FUNCTION_BLOCK FB_CameraTrigger EXTENDS FB_Commons IMPLEMENTS I_CameraTrigger, I_StartPosDetect
(*************************************************************************************************)
(*  FILENAME:    FB_CameraTrigger                                                                *)
(*  PROJECT:     CALMAR PUPLC                                                                    *)
(*  COPYRIGHT:   All rights reserved (c) Wifag//Polytype, Fribourg/Switzerland (2016)            *)
(*  ENVIRONMENT: TwinCAT PLC                                                                     *)
(*  VERSION:     <version>                                                                       *)
(*************************************************************************************************)
(*  DESCRIPTION:                                                                   <description> *)
(*    Generate timestamp trigger output based on timestamp sensor input. Two variants            *)
(*    exist, a timebased approach where the trigger time is calculated at the time the sensor    *)
(*    event occurs, and a second approach where the sensor event time is translated to a sensor  *)
(*    event position, and a trigger is generated when the calculated trigger position has almost *)
(*    been reached. The second approach has the advantage that is is less susceptible to speed   *)
(*    variations.                                                                                *)
(*                                                                                </description> *)
(*************************************************************************************************)

{library public}
VAR_INPUT
  bI_HwEnable                             : BOOL;            // relase (enable SheetDetect) from machine
  (* - (EL1252) StartPosition detect sensor*)
  bI_Sensor_State                   AT%I* : BOOL;            // Sensor signal
  tI_Sensor_TimeStampPos            AT%I* : T_DCTIME64;      // Sensor last detection timestamp
  (* - (EL1252) Camera started feedback trigger/signal*)
  bI_TriggerFeedback_State          AT%I* : BOOL;           // Sensor signal
  tI_TriggerFeedback_TimeStampPos   AT%I* : T_DCTIME64;     // Sensor last detection timestamp

  (*System signals*)
  iI_CurrentPos                   : DINT;                   // Current position in [SubPx]*)
  fI_ConveyorSpeed                : LREAL;                  // Current speed of substrate in [m/s]*)
  
  (*Exernal command*)
 // bI_ManualTeach                  : BOOL;                   // External manual teach is active

  (*Debug & Test*)
  bI_ManualTrigger                : BOOL;                   // Manual start trigger
END_VAR

VAR_OUTPUT
  (*Link to EL2252*)
  ObTrigger                 AT%Q* : BOOL;                   // EL2252 Output1 - TRUE=start camer
  OtTriggerStartTime        AT%Q* : T_DCTIME64;             // EL2252 Timestamp - where to set outputs
  OnTriggerCommand          AT%Q* : BYTE;                   // EL2252 Command - activation timestamp ouput
END_VAR

(*{library private}*)
VAR
  bInitOk                         : BOOL;           // initialized
  bSpeedValid                     : BOOL;           // speed is valid
  bTriggerArmed                   : BOOL;           // trigger is armed
  bCamValid                       : BOOL;           // camera is valid
  bTriggerOk                      : BOOL;
  rT_Sensor                       : R_TRIG;        // rising edge trigger sensor
  
  (*configuration*)
  _nResolution                    : INT := 1;       // Printhead Resolution [e.g. 600] x Subpixel Resolution [e.g. 32]*)
  _bUsePositionTrigger            : BOOL;           // FALSE: Calculate time with speed and position distance@sensor event, TRUE: Calculate sensor event position, launch trigger based on position
  _bUseCameraTrigger              : BOOL;           // (cam specific setting) Generate camera trigger output
  _bUseCameraTriggerFeedback      : BOOL;           // (cam specific setting) Evaluate camera triggered feedback
  _bCamManualTeachMode            : BOOL;           // cam in manual teach mode
  _tMemTriggerFeedback_TimeStampPos : T_DCTIME64;
  _nSubstrateLength               : DINT;           // Substrate length in pulse [SubPx]
  _fSubstrateLength               : LREAL;          // Substrate length in [m]
  _fTriggerDistance               : LREAL;          // Distance between Sensor and Trigger [m]
  _fTriggerLength                 : LREAL := 10;    // Length of trigger signal in ms, min. 3 bus cycles
  
  iActiveCam	                    : I_CameraTriggerDevice;  // active camera interface
  
  bSheetDetected                  : BOOL;
  bInhibitTrigger                 : BOOL;            (*inhibit trigger signals, TRUE=inhibit*)
  bReleaseInhibitTrigger          : BOOL;            (*condition to release inhibit trigger*)

  eState                          : BYTE;            (*State*)
  tSensor_TimeStamp               : T_DCTIME64;      (*Sensor last detection timestamp*)
  tTriggerFeedback_TimeStamp      : T_DCTIME64;      (*Trigger feedback last detection timestamp*)
  tCurrentTime                    : T_DCTIME64;      (*Current system dc time [64bit]*)
  tTrigger_EventTime              : T_DCTIME64;      (*Trigger event timestamp*)

  _bManualStart                   : BOOL;
  fDeltaDistance                  : LREAL;           (*Distance that the substrate moved between the detection and the treatment of the information [m]*)
  _nX0                            : DINT;            (*Detected X0 position of CT [SubPx] by sensor*)
  _nCamStartPos                   : DINT;            (*Camera start position*)
  _nCamStartedPos                 : DINT;            (*Camera started position [SubPx]*)
  
  tCurrentTimeStamp               : T_DCTIME64;      (* Get Current Timestamp *)
  tLastTimeStamp                  : T_DCTIME64;      (* Get Current Timestamp *)
  fCycleTime                      : LREAL;           (* Current calcualted cycle time [s]*)

  fRemDist                        : LREAL;           (*Remaining distance until trigger occurs [m]*)
  fPreTriggerPosition             : LREAL;           (*Margin between effective trigger position and generation of timestamp*)

  fb_FTrig_ManualTeach            : F_TRIG;          (*FTrig for teach to release inhibit*)
  
  (*Debug*)
  _bVerbose                       : BOOL;
END_VAR

VAR CONSTANT
  fC_MIN_CONVEYOR_SPEED           : LREAL := 0.01;
  fC_PreTrigFactor                : LREAL := 3.0;
  fC_SheetLengthMargin            : LREAL := 0.01;   (*Added 10 mm margin for substrate length in case of print quality strips at the end of sheet in case of start with edge*)
  fC_MaxCameraFeedbackTimeout     : LREAL := 28.0;   (*[ns] Max. timeout waiting for camera trigger feedback signal*)

  (*State*)
  cL_IDLE                         : BYTE := 0;       (*Idle state, no trigger active*)
  cL_SENSOREVENT                  : BYTE := 1;       (*Sensor started trigger generation*)
  cL_WAITALMOSTSTART              : BYTE := 2;       (*Wait timestamp calculation critera*)
  cL_WAITSTART                    : BYTE := 3;       (*Wait for trigger generation critera*)
  cL_WAITFEEDBACK                 : BYTE := 4;       (*Wait on feedback from trigger*)
  cL_TRIGACTIVE                   : BYTE := 5;       (*Trigger set*)
  cL_WAITSTOP                     : BYTE := 6;       (*Trigger reset*)

  (*EL2252 Command*)
  cL_INACTIVE                     : BYTE := 0;
  cL_ACTIVE                       : BYTE := 3;
END_VAR
// TODO: convert all LREAL_TO_ULINT to save functions with range overflow check (add to CalmarCommons) to prevent crashes

IF NOT bInitOk THEN RETURN; END_IF;

// General calculations
bSpeedValid   := fI_ConveyorSpeed > fC_MIN_CONVEYOR_SPEED;    // speed valid (ignore trigger if not moving)
bCamValid     := SEL(iActiveCam<>0, FALSE, TRUE);             // camera valid (ignore trigger otherwise)
tCurrentTime  := F_GetCurDcTaskTime64();                      // current dc time (most accurate time stamp we have)
fCycleTime    := (TO_LREAL(tCurrentTime) - TO_LREAL(tLastTimeStamp)) * 1E-9;  tLastTimeStamp  := tCurrentTime;  // calculate cycle time of this block
bSheetDetected:= FALSE;                                       // Set to true below just for one cycle
bTriggerArmed :=  NOT bInhibitTrigger AND bSpeedValid AND bI_HwEnable;
rT_Sensor(CLK:=bI_Sensor_State);

IF bCamValid THEN    // save dynamic changable settings
  _fTriggerDistance := iActiveCam.fTriggerDistance;
  _fTriggerLength   := iActiveCam.fTriggerPulseLength;
END_IF


(*State Machine ----------------------------------------------------------------*)
CASE eState OF
  cL_IDLE:     (*Not started, waiting for start trigger*)
  
    IF bTriggerArmed THEN (*ignore trigger else*)
 
      IF rT_Sensor.Q AND (bCamValid OR _bCamManualTeachMode) THEN      (*Start launched*)
        eState            := cL_SENSOREVENT;
        tSensor_TimeStamp := tI_Sensor_TimeStampPos;
        _bManualStart := FALSE;
        IF _bCamManualTeachMode THEN LogWarning('StartTrigger in manual teach mode'); END_IF
      ELSIF (bI_ManualTrigger AND bCamValid) THEN  (*Manual start launched*)
        eState            := cL_SENSOREVENT;
        tSensor_TimeStamp := tCurrentTime;
        _bManualStart := TRUE;
      ELSIF (rT_Sensor.Q OR bI_ManualTrigger) AND NOT bCamValid THEN   (*Trigger without active camera*)
        LogWarning('No camera or start device active, ignore trigger');
      END_IF;
      
    END_IF
    
    OnTriggerCommand := cL_INACTIVE;
    ObTrigger        := FALSE;

  cL_SENSOREVENT:     (*Not started*)
    IF NOT bSpeedValid THEN 
      eState := cL_IDLE;        // ignore trigger if not moving anymore (avoid zero division)
    ELSE
      (*Distance in [m] that the substrate has traveled between the sensor detection (time) current plc cycle*)
      fDeltaDistance     := UINT64_TO_LREAL(UInt64Sub64(ULINT_TO_ULARGE(tCurrentTime), ULINT_TO_ULARGE(tSensor_TimeStamp))) * 1E-9 * fI_ConveyorSpeed;
      (*Position where the sheet has been detected in [SubPx]*)
      _nX0               := iI_CurrentPos - F_MeterToSubPixel(fPosMeter:=fDeltaDistance, fResoSubPx:=_nResolution);
      
      IF _bUsePositionTrigger OR NOT _bUseCameraTrigger THEN
        eState             := cL_WAITALMOSTSTART;
      ELSE
        eState             := cL_WAITSTART;
        tTrigger_EventTime := (tSensor_TimeStamp + LREAL_TO_ULINT(_fTriggerDistance / fI_ConveyorSpeed * 1E9));
      END_IF;
      
      OnTriggerCommand := cL_INACTIVE;
      ObTrigger         := TRUE;
      bInhibitTrigger   := TRUE;
      bSheetDetected    := TRUE;
      
    END_IF

  cL_WAITALMOSTSTART: (*Only active when bI_UsePositionTrigger=TRUE: wait until Start position almost reached, then set timestamp*)
    (*Remaining distance in [m], converted to REAL to avoid integer wrap problems*)
    fRemDist             := _fTriggerDistance + (DINT_TO_REAL(_nX0) - DINT_TO_REAL(iI_CurrentPos))*0.0254 / INT_TO_REAL(_nResolution);
    fPreTriggerPosition  := fC_PreTrigFactor * fCycleTime * fI_ConveyorSpeed;

    IF fRemDist < fPreTriggerPosition THEN
      eState             := cL_WAITSTART;
      tTrigger_EventTime := (tSensor_TimeStamp + LREAL_TO_ULINT(fRemDist / fI_ConveyorSpeed * 1E9));    // division save because we are moving to reach this position
      IF _bUseCameraTrigger AND NOT _bManualStart THEN
        OnTriggerCommand := cL_ACTIVE;  (*Arm EL2252*)
      END_IF
      LogTsDiff(aIdent:= 'WAITALMOSTSTART: ', t1:=tTrigger_EventTime, t2:=tCurrentTime);
    ELSE
      eState           := cL_WAITALMOSTSTART;
      OnTriggerCommand := cL_INACTIVE;
    END_IF;
    ObTrigger          := TRUE;

  cL_WAITSTART:       (*Wait until start time reached*)
    bTriggerOk := TRUE;
    IF (tTrigger_EventTime < tCurrentTime) THEN (* StartTime elapsed *)
      // position reached
      IF _bUseCameraTriggerFeedback THEN
        eState         := cL_WAITFEEDBACK;
      ELSE
        eState         := cL_TRIGACTIVE;
        iActiveCam.CamTrigger(bOk:=bTriggerOk, nPos:=iI_CurrentPos, nPosDeviation:=0);
      END_IF

      OnTriggerCommand := cL_INACTIVE; (*Disarm already command to EL2252, trigger generated*)
    ELSE
      // position not yet reached
      eState           := cL_WAITSTART;
      IF _bUseCameraTrigger AND NOT _bManualStart THEN
        OnTriggerCommand := cL_ACTIVE;  (*Arm EL2252*)
      END_IF
    END_IF;

    ObTrigger      := TRUE;  
    
  cL_WAITFEEDBACK:
    IF _bManualStart THEN //Simulate feedback in case of manual start
      tTriggerFeedback_TimeStamp:= tTrigger_EventTime + LREAL_TO_ULINT(1000.0 * 1E3); //Trigger event plus 1000ns
    ELSE
      IF tI_TriggerFeedback_TimeStampPos = _tMemTriggerFeedback_TimeStampPos AND tCurrentTime > (tTrigger_EventTime + LREAL_TO_ULINT(fC_MaxCameraFeedbackTimeout * 1E3)) THEN
        // feedback was not received in next plc cycle (timeout jitter in camera max. 28us)
        LogError(F_Concat3('No Camera trigger feedback received (timeout), after ', TO_STRING(TO_LREAL(tCurrentTime-tTrigger_EventTime)/1E6), 'ms'));
        bTriggerOk := FALSE;
        tTriggerFeedback_TimeStamp:= tTrigger_EventTime + LREAL_TO_ULINT(fC_MaxCameraFeedbackTimeout * 1E3);
      ELSE
        tTriggerFeedback_TimeStamp:= tI_TriggerFeedback_TimeStampPos;
			END_IF
    END_IF
    
  (*feedback signal is a very short trigger that the PLC sometimes cannot register, therefore we use the timestamp*)
    IF (tTriggerFeedback_TimeStamp <> _tMemTriggerFeedback_TimeStampPos) AND (tTriggerFeedback_TimeStamp > 0) OR _bManualStart THEN
      eState          := cL_TRIGACTIVE;
      // start position requested
      fDeltaDistance  := UINT64_TO_LREAL(UInt64Sub64(ULINT_TO_ULARGE(tCurrentTime), ULINT_TO_ULARGE(tTrigger_EventTime))) * 1E-9 * fI_ConveyorSpeed;
      _nCamStartPos   := _nX0 +   F_MeterToSubPixel(fPosMeter:=_fTriggerDistance, fResoSubPx:=_nResolution);
      
      // effective started position
      fDeltaDistance  := UINT64_TO_LREAL(UInt64Sub64(ULINT_TO_ULARGE(tCurrentTime), ULINT_TO_ULARGE(tTriggerFeedback_TimeStamp))) * 1E-9 * fI_ConveyorSpeed;
      _nCamStartedPos := iI_CurrentPos - F_MeterToSubPixel(fPosMeter:=fDeltaDistance, fResoSubPx:=_nResolution);
      IF _bManualStart THEN iActiveCam.CamTrigger(bOk:=bTriggerOk, nPos:=_nCamStartPos, nPosDeviation:=0);
      ELSE                  iActiveCam.CamTrigger(bOk:=bTriggerOk, nPos:=_nCamStartPos, nPosDeviation:=-_nCamStartedPos+_nCamStartPos); END_IF  (*!!!!   sign inverted*)
    ELSE
     eState           := cL_WAITFEEDBACK;
    END_IF    
    
  cL_TRIGACTIVE:   (*Trigger high*)
    eState         := cL_WAITSTOP;
    
    // calculate end timestamp of trigger (end of trigger active signal)
    tTrigger_EventTime := (tTrigger_EventTime + LREAL_TO_ULINT(_fTriggerLength * 1E6));
    
    OnTriggerCommand := cL_INACTIVE;
    ObTrigger        := FALSE;
    
  cL_WAITSTOP:  (*Wait until trigger time has elapsed*)
    IF (tTrigger_EventTime < tCurrentTime) THEN (* StopTime elapsed *)
      eState           := cL_IDLE;
      OnTriggerCommand := cL_INACTIVE; (*Disarm EL2252, trigger generated*)
      iActiveCam.CamTriggerDone();
    ELSE
      eState           := cL_WAITSTOP;
      IF _bUseCameraTrigger THEN
        OnTriggerCommand := cL_ACTIVE;  (*Arm EL2252*)
      END_IF
    END_IF;

    ObTrigger        := FALSE;

  ELSE  (*Default*)
    eState           := cL_IDLE;
    ObTrigger        := FALSE;
    OnTriggerCommand := cL_INACTIVE;
END_CASE;

OtTriggerStartTime := tTrigger_EventTime;

_tMemTriggerFeedback_TimeStampPos := tI_TriggerFeedback_TimeStampPos;

(*Release inhibit trigger*)
bReleaseInhibitTrigger := (iI_CurrentPos >= (_nX0 + _nSubstrateLength));
//fb_FTrig_ManualTeach(CLK := bI_ManualTeach);

IF (bReleaseInhibitTrigger OR fb_FTrig_ManualTeach.Q) AND bInhibitTrigger THEN
	bInhibitTrigger := FALSE;
END_IF;

(********************************* END OF FB *****************************************************)

PROPERTY bManualTeach : BOOL
GET
bManualTeach := _bCamManualTeachMode;
END_GET
SET
_bCamManualTeachMode := bManualTeach;
END_SET
END_PROPERTY

(*
  A new container detected on X0.
  NOTE: a pulse only
*)
PROPERTY bStartTrig : BOOL
GET
bStartTrig := bSheetDetected;
END_GET
END_PROPERTY

(*
  A valid container detected.
*)
PROPERTY bValid : BOOL
GET
bValid := bSheetDetected AND NOT _bCamManualTeachMode AND bCamValid;  // in manual teach the ct is "present" should not be printed
END_GET
END_PROPERTY

METHOD Disable : BOOL
IF eState = cL_IDLE THEN
  iActiveCam := 0;
  Disable := TRUE;
ELSE  
  Disable := FALSE;
  LogError('disable failed: trigger busy');
END_IF
END_METHOD

METHOD Enable : BOOL
VAR_INPUT
	iCam	                    : I_CameraTriggerDevice;
  bUseCameraTrigger         : BOOL; //Generate camera trigger
  bUseCameraTriggerFeedback : BOOL; //Use feedback as trigger?
END_VAR
IF iCam = 0 THEN
  Enable := FALSE;
  LogError('setCam failed: invalid reference');
ELSIF eState <> cL_IDLE THEN
  Enable := FALSE;
  LogError('enable failed: trigger busy');
ELSE
  iActiveCam := iCam;
  Enable     := TRUE;

  // save constant settings
  _bUseCameraTrigger := bUseCameraTrigger;
  _bUseCameraTriggerFeedback := bUseCameraTriggerFeedback;
END_IF;
END_METHOD

METHOD Init
VAR_INPUT
  nResolution                   : INT := 1;        (*Printhead Resolution [e.g. 600] x Subpixel Resolution [e.g. 32]*)
  bUsePositionTrigger           : BOOL;            (*FALSE: Calculate time with speed and position distance@sensor evont*)
END_VAR
(*zero divisions*)
IF nResolution = 0 THEN 
  bInitOk :=FALSE;
  RETURN; 
END_IF;

_nResolution:=nResolution;
_bUsePositionTrigger :=bUsePositionTrigger;


bInitOk :=TRUE;
END_METHOD

(*
  Log timestamp difference (if verbose active).
  t1-t2 
*)
METHOD LogTsDiff : BOOL
VAR_INPUT
  aIdent : STRING;
  t1 : T_DCTIME64;
  t2 : T_DCTIME64;
END_VAR
IF _bVerbose THEN
  LogLvl(Lvl:=E_LogSeverity.Debug, Msg:=
       F_Concat7(aIdent, 
                 't1: ', TO_STRING(t1), 
                 ' t2: ', TO_STRING(t2), 
                 ' t1-t2 [ms]: ', TO_STRING((TO_LREAL(t1)-TO_LREAL(t2))*1E-6)
       )
  );
END_IF
END_METHOD

(*
  Detected start position X0 (absolute) in [SubPx].
*)
PROPERTY nStartPositionX0 : DINT
GET
nStartPositionX0 := _nX0;
END_GET
END_PROPERTY

METHOD Reset
VAR_INPUT
END_VAR
eState          := cL_IDLE;
bInhibitTrigger := FALSE;
END_METHOD

METHOD SetSubstrateLength
VAR_INPUT
  fSubstrateLength : LREAL;
END_VAR
IF NOT bInitOk THEN RETURN;END_IF;

(*Added 10 mm margin for substrate length in case of print quality strips at the end of sheet in case of start with edge*)
_fSubstrateLength := fSubstrateLength + fC_SheetLengthMargin;
_nSubstrateLength := F_MeterToSubPixel(fPosMeter:=_fSubstrateLength, fResoSubPx:=_nResolution);
END_METHOD

END_FUNCTION_BLOCK

(* stored: Version 1.1.0.1, ProductVersion 3.1.4024.3
   POU FB_CameraTrigger: Id {b0f3b9ca-3ef5-425e-9c4d-fa0358aa72fd}, SpecialFunc None
   Property bManualTeach: Id {58f64ca5-2fbd-4f19-9c85-e284ce94b427}
   Get Get: Id {4c3cab32-2be9-4a94-8004-e45185b9890b}
   Set Set: Id {7bf6ee58-08a2-435d-af4d-9a1743824b8f}
   Property bStartTrig: Id {744708b2-efbe-44a0-b99d-f740e061c41a}
   Get Get: Id {b18ba1e7-5e2d-475f-8323-33bbcd1c692c}
   Property bValid: Id {b121f0c2-19e1-4824-90fe-d08dc84adecf}
   Get Get: Id {0213548a-6652-4f40-88ae-053b91249e4e}
   Method Disable: Id {8de1e61a-7ae8-4635-898a-17c0e033e723}
   Method Enable: Id {3a388c10-901b-466a-867e-ff1154655991}
   Method Init: Id {df11c7a2-a5d2-4167-96a4-15a760cac9c3}
   Method LogTsDiff: Id {998b1383-3728-46bb-839b-a9a799ecec56}
   Property nStartPositionX0: Id {c9eb7bc9-f55d-4283-bb08-a90d79e764fa}
   Get Get: Id {259de372-e988-4571-a3a2-e4601c5b4a52}
   Method Reset: Id {c3f1176f-9f21-4574-a83d-31acfd8f4d0c}
   Method SetSubstrateLength: Id {5205cec1-13bd-4eb7-92d4-8661d94d2b89} *)
